TYPE ST_ControllerStatus :
STRUCT
	ControllerOn		: BOOL;
	SelfOptimization	: BOOL;
	ManualMode			: BOOL;
	SetpointSwitch		: BOOL;
	OptimizationError	: BOOL;
	DataNotValid		: BOOL;
	Overload			: BOOL;
	NetOverload			: BOOL;
END_STRUCT
END_TYPE

(* stored: Version 1.1.0.1, ProductVersion 3.1.4024.16
   DUT ST_ControllerStatus: Id {fb7d768b-9ece-0aa5-0133-5713c70e8b26} *)
